// TwinCAT 3 PLC project PLC_Dev_Anker1
// ProgramVersion: 3.1.4024.0
// libraries:
//   EfficientIO Communicator, * (EfficientIO)
//   Tc2_Standard, * (Beckhoff Automation GmbH)
//   Tc2_System, * (Beckhoff Automation GmbH)
//   Tc3_Module, * (Beckhoff Automation GmbH)
// project tree:
//   DUTs/ struct_ADS_Anker.TcDUT
//   / FastTask.TcTTO, MiddleTask.TcTTO, SlowTask.TcTTO
//   FB/ FB_ADS_Read.TcPOU, F_AdsErrorText.TcPOU
//   POUs/ prgComEffIO.TcPOU, prgEM.TcPOU, prgEMS.TcPOU, prgRWEffIO.TcPOU, prgVarEffIO.TcPOU, prg_ADS.TcPOU
// (motion and I/O tree: see PLC project plc dev barac)
// real-time tasks:
//   TASK FastTask: cycle T#5ms, priority 19, ADS port 351
//   TASK SlowTask: cycle T#20ms, priority 22, ADS port 352
//   TASK MiddleTask: cycle T#10ms, priority 21, ADS port 353

CONFIGURATION PLC_Dev_Anker1
    RESOURCE PLC ON TwinCAT3
        TASK FastTask(INTERVAL := T#5ms, PRIORITY := 19);
        TASK MiddleTask(INTERVAL := T#10ms, PRIORITY := 21);
        TASK SlowTask(INTERVAL := T#20ms, PRIORITY := 22);
        PROGRAM prgRWEffIO WITH FastTask : prgRWEffIO;
        PROGRAM prgVarEffIO WITH FastTask : prgVarEffIO;
        PROGRAM prgEMS WITH MiddleTask : prgEMS;
        PROGRAM prgEM WITH MiddleTask : prgEM;
        PROGRAM prg_ADS WITH MiddleTask : prg_ADS;
        PROGRAM prgComEffIO WITH SlowTask : prgComEffIO;
    END_RESOURCE
END_CONFIGURATION

// ---- DUTs/struct_ADS_Anker.TcDUT
TYPE struct_ADS_Anker :
STRUCT
	int_liveCount		: INT;	
	
	// prgEM
	lr_RealPower_Grid			: LREAL;				
	lr_ApparentPower_Grid		: LREAL;				
	lr_ReactivePower_Grid		: LREAL;				
	lr_Frequency_Grid			: LREAL;				                                   
	lr_Voltage_L1N				: LREAL;				
	lr_Voltage_L2N				: LREAL;				
	lr_Voltage_L3N				: LREAL;				
	lr_Voltage_L1L2				: LREAL;				
	lr_Voltage_L2L3				: LREAL;				
	lr_Voltage_L3L1				: LREAL;				
 	lr_Current_L1				: LREAL;				
	lr_Current_L2				: LREAL;				
	lr_Current_L3				: LREAL;				
	lrPower_EM1					: LREAL;					
	lrPower_EM2					: LREAL;					
	lrPower_EM3					: LREAL;					
	lrPower_EM4					: LREAL;					
	lrPower_EM5					: LREAL;					
	lrPower_EM6					: LREAL;					
	lrPower_House				: LREAL;					
	lr_EnergyCounter_Grid		: LREAL;					
	lr_EnergyCounter_EM1		: LREAL;					
	lr_EnergyCounter_EM2		: LREAL;					
	lr_EnergyCounter_EM3		: LREAL;					
	lr_EnergyCounter_EM4		: LREAL;					
	lr_EnergyCounter_EM5		: LREAL;					
	lr_EnergyCounter_EM6		: LREAL;					
	lr_EnergyCounter_House		: LREAL;		

	// prgEMS
	b_Manual_On_CH1				: BOOL;						
	b_Manual_Off_CH1			: BOOL;						
	b_Manual_On_CH2				: BOOL;						
	b_Manual_Off_CH2			: BOOL;						
	b_Manual_On_CH3				: BOOL;						
	b_Manual_Off_CH3			: BOOL;						
	b_Manual_On_CH4				: BOOL;						
	b_Manual_Off_CH4			: BOOL;						
	b_Manual_On_CH5				: BOOL;						
	b_Manual_Off_CH5			: BOOL;						
	b_Manual_On_Coffee_CH6		: BOOL;				
	b_Manual_Off_Coffee_CH6		: BOOL;				
	b_Manual_On_Vent_CH7		: BOOL;				
	b_Manual_Off_Vent_CH7		: BOOL;			
	b_LoadOn_CH1				: BOOL;		
	b_LoadOn_CH2				: BOOL;			
	b_LoadOn_CH3				: BOOL;			
	b_LoadOn_CH4				: BOOL;			
	b_LoadOn_CH5				: BOOL;			
	b_LoadOn_CH6				: BOOL;			
	b_LoadOn_CH7				: BOOL;		
	byte_MoFr_Open_Hour			: BYTE;					
	byte_MoFr_Open_Minute		: BYTE;					
	byte_MoFr_Close_Hour		: BYTE;					
	byte_MoFr_Close_Minute		: BYTE;					
	byte_Sa_Open_Hour			: BYTE;					
	byte_Sa_Open_Minute			: BYTE;					
	byte_Sa_Close_Hour			: BYTE;					
	byte_Sa_Close_Minute		: BYTE;					
	byte_So_Open_Hour			: BYTE;					
	byte_So_Open_Minute			: BYTE;					
	byte_So_Close_Hour			: BYTE;					
	byte_So_Close_Minute		: BYTE;					
// offset CH1 in hours			                    
	b_Enable_Control_CH1		: BOOL;				
	real_Offset_Start_CH1		: REAL;				
	real_Offset_Stop_CH1		: REAL;				
// offset CH2 in hours			                    
	b_Enable_Control_CH2		: BOOL;				
	real_Offset_Start_CH2		: REAL;				
	real_Offset_Stop_CH2		: REAL;				
// offset CH3 in hours			                    
	b_Enable_Control_CH3		: BOOL;				
	real_Offset_Start_CH3		: REAL;				
	real_Offset_Stop_CH3		: REAL;				
// offset CH4 in hours			                    
	b_Enable_Control_CH4		: BOOL;				
	real_Offset_Start_CH4		: REAL;				
	real_Offset_Stop_CH4		: REAL;				
// offset CH5 in hours			                    
	b_Enable_Control_CH5		: BOOL;				
	real_Offset_Start_CH5		: REAL;				
	real_Offset_Stop_CH5		: REAL;				
// offset CH6 in hours			                    
	b_Enable_Control_Coffee_CH6	: BOOL;				
	real_Offset_Start_Coffee_CH6: REAL;				
	real_Offset_Stop_Coffee_CH6	: REAL;				
// offset CH7 in hours			                    
	b_Enable_Control_Vent_CH7	: BOOL;				
	real_Offset_Start_CH7		: REAL;				
	real_Offset_Stop_CH7		: REAL;				


                                  
			(*: REAL;			                        
			: REAL;                                     
			: REAL;			
			: REAL;			
			: REAL;
			: REAL;			
			: REAL;
			: REAL;			
*)

END_STRUCT
END_TYPE

// ---- POUs/prgRWEffIO.TcPOU
PROGRAM prgRWEffIO
VAR
	fbRW1		: FB_ReadWrite_V2;
END_VAR

fbRW1(eUploadType := eSelectDataUploadType.e_Change_Intervall5min, bBusy=> , bError=> , udiErrorCodeOut=> , eErrorReadWrite_Out=> );

END_PROGRAM

// ---- POUs/prgVarEffIO.TcPOU
PROGRAM prgVarEffIO
VAR
	fbVar		: FB_VarInfo_V3;
END_VAR

fbVar(
	bReadInfo:= , 
	eTMCFile:= eSelectTMCFile.eDontUseTMCFile, 
	eSavePositionTMCFile:= eSavePositionOnPLC.ePostionC, 
	udiCounterFoundVariables=> , 
	bError=> , 
	bBusy=> , 
	byProgress=> , 
	udiErrorCodeOut=> , 
	eErrorVarInfo_Out=> , 
	sVarWithError=> );

fbVar(
	bReadInfo:= , 
	eTMCFile:= eSelectTMCFile.eDontUseTMCFile, 
	eSavePositionTMCFile:= eSavePositionOnPLC.ePostionC,
	udiCounterFoundVariables=> , 
	bError=> , 
	bBusy=> , 
	byProgress=> , 
	udiErrorCodeOut=> , 
	eErrorVarInfo_Out=> , 
	sVarWithError=> );
	
fbVar(
	bReadInfo:= , 
	eTMCFile:= eSelectTMCFile.eDontUseTMCFile, 
	eSavePositionTMCFile:= eSavePositionOnPLC.ePostionC,
	udiCounterFoundVariables=> , 
	bError=> , 
	bBusy=> , 
	byProgress=> , 
	udiErrorCodeOut=> , 
	eErrorVarInfo_Out=> , 
	sVarWithError=> );

END_PROGRAM

// ---- POUs/prgEMS.TcPOU
PROGRAM prgEMS
VAR	
	b_Manual_On_CH1		: BOOL;						//{#lynus.ag#()}
	b_Manual_Off_CH1	: BOOL;						//{#lynus.ag#()}
	b_Manual_On_CH2		: BOOL;						//{#lynus.ag#()}
	b_Manual_Off_CH2	: BOOL;						//{#lynus.ag#()}
	b_Manual_On_CH3		: BOOL;						//{#lynus.ag#()}
	b_Manual_Off_CH3	: BOOL;						//{#lynus.ag#()}
	b_Manual_On_CH4		: BOOL;						//{#lynus.ag#()}
	b_Manual_Off_CH4	: BOOL;						//{#lynus.ag#()}
	b_Manual_On_CH5		: BOOL;						//{#lynus.ag#()}
	b_Manual_Off_CH5	: BOOL;						//{#lynus.ag#()}
	b_Manual_On_Coffee_CH6		: BOOL;						//{#lynus.ag#()}
	b_Manual_Off_Coffee_CH6		: BOOL;						//{#lynus.ag#()}
	b_Manual_On_Vent_CH7		: BOOL;						//{#lynus.ag#()}
	b_Manual_Off_Vent_CH7		: BOOL;						//{#lynus.ag#()}
	mtest: BOOL;

	b_LoadOn_CH1	: BOOL;						//{#lynus.ag#()}
	b_LoadOn_CH2	: BOOL;						//{#lynus.ag#()}
	b_LoadOn_CH3	: BOOL;						//{#lynus.ag#()}
	b_LoadOn_CH4	: BOOL;						//{#lynus.ag#()}
	b_LoadOn_CH5	: BOOL;						//{#lynus.ag#()}
	b_LoadOn_CH6	: BOOL;						//{#lynus.ag#()}
	b_LoadOn_CH7	: BOOL;						//{#lynus.ag#()}
	b_Input_KeySwitch		: BOOL;						//{#lynus.ag#()}
	b_Input_Spare			: BOOL;						//{#lynus.ag#()}
	m_UnderGroundMode		: BOOL;						//{#lynus.ag#()}
// opening hours
	byte_MoFr_Open_Hour		:BYTE;					//{#lynus.ag#()}
	byte_MoFr_Open_Minute	:BYTE;					//{#lynus.ag#()}
	byte_MoFr_Close_Hour	:BYTE;					//{#lynus.ag#()}
	byte_MoFr_Close_Minute	:BYTE;					//{#lynus.ag#()}
	byte_Sa_Open_Hour		:BYTE;					//{#lynus.ag#()}
	byte_Sa_Open_Minute		:BYTE;					//{#lynus.ag#()}
	byte_Sa_Close_Hour		:BYTE;					//{#lynus.ag#()}
	byte_Sa_Close_Minute	:BYTE;					//{#lynus.ag#()}
	byte_So_Open_Hour		:BYTE;					//{#lynus.ag#()}
	byte_So_Open_Minute		:BYTE;					//{#lynus.ag#()}
	byte_So_Close_Hour		:BYTE;					//{#lynus.ag#()}
	byte_So_Close_Minute	:BYTE;					//{#lynus.ag#()}
// offset CH1 in hours			
	b_Enable_Control_CH1		:BOOL;				//{#lynus.ag#()}
	real_Offset_Start_CH1		:REAL;				//{#lynus.ag#()}
	real_Offset_Stop_CH1		:REAL;				//{#lynus.ag#()}
// offset CH2 in hours			
	b_Enable_Control_CH2		:BOOL;				//{#lynus.ag#()}
	real_Offset_Start_CH2		:REAL;				//{#lynus.ag#()}
	real_Offset_Stop_CH2		:REAL;				//{#lynus.ag#()}
// offset CH3 in hours			
	b_Enable_Control_CH3		:BOOL;				//{#lynus.ag#()}
	real_Offset_Start_CH3		:REAL;				//{#lynus.ag#()}
	real_Offset_Stop_CH3		:REAL;				//{#lynus.ag#()}
// offset CH4 in hours			
	b_Enable_Control_CH4		:BOOL;				//{#lynus.ag#()}
	real_Offset_Start_CH4		:REAL;				//{#lynus.ag#()}
	real_Offset_Stop_CH4		:REAL;				//{#lynus.ag#()}
// offset CH5 in hours			
	b_Enable_Control_CH5		:BOOL;				//{#lynus.ag#()}
	real_Offset_Start_CH5		:REAL;				//{#lynus.ag#()}
	real_Offset_Stop_CH5		:REAL;				//{#lynus.ag#()}
// offset CH6 in hours			
	b_Enable_Control_Coffee_CH6	:BOOL;				//{#lynus.ag#()}
	real_Offset_Start_Coffee_CH6:REAL;				//{#lynus.ag#()}
	real_Offset_Stop_Coffee_CH6	:REAL;				//{#lynus.ag#()}
// offset CH7 in hours			
	b_Enable_Control_Vent_CH7	:BOOL;				//{#lynus.ag#()}
	real_Offset_Start_CH7		:REAL;				//{#lynus.ag#()}
	real_Offset_Stop_CH7		:REAL;				//{#lynus.ag#()}
END_VAR

b_Manual_On_CH1	:=	prg_ADS.struct_received.b_Manual_On_CH1	;
b_Manual_Off_CH1	:=	prg_ADS.struct_received.b_Manual_Off_CH1	;
b_Manual_On_CH2	:=	prg_ADS.struct_received.b_Manual_On_CH2	;
b_Manual_Off_CH2	:=	prg_ADS.struct_received.b_Manual_Off_CH2	;
b_Manual_On_CH3	:=	prg_ADS.struct_received.b_Manual_On_CH3	;
b_Manual_Off_CH3	:=	prg_ADS.struct_received.b_Manual_Off_CH3	;
b_Manual_On_CH4	:=	prg_ADS.struct_received.b_Manual_On_CH4	;
b_Manual_Off_CH4	:=	prg_ADS.struct_received.b_Manual_Off_CH4	;
b_Manual_On_CH5	:=	prg_ADS.struct_received.b_Manual_On_CH5	;
b_Manual_Off_CH5	:=	prg_ADS.struct_received.b_Manual_Off_CH5	;
b_Manual_On_Coffee_CH6	:=	prg_ADS.struct_received.b_Manual_On_Coffee_CH6	;
b_Manual_Off_Coffee_CH6	:=	prg_ADS.struct_received.b_Manual_Off_Coffee_CH6	;
b_Manual_On_Vent_CH7	:=	prg_ADS.struct_received.b_Manual_On_Vent_CH7	;
b_Manual_Off_Vent_CH7	:=	prg_ADS.struct_received.b_Manual_Off_Vent_CH7	;
b_LoadOn_CH1	:=	prg_ADS.struct_received.b_LoadOn_CH1	;
b_LoadOn_CH2	:=	prg_ADS.struct_received.b_LoadOn_CH2	;
b_LoadOn_CH3	:=	prg_ADS.struct_received.b_LoadOn_CH3	;
b_LoadOn_CH4	:=	prg_ADS.struct_received.b_LoadOn_CH4	;
b_LoadOn_CH5	:=	prg_ADS.struct_received.b_LoadOn_CH5	;
b_LoadOn_CH6	:=	prg_ADS.struct_received.b_LoadOn_CH6	;
b_LoadOn_CH7	:=	prg_ADS.struct_received.b_LoadOn_CH7	;
byte_MoFr_Open_Hour	:=	prg_ADS.struct_received.byte_MoFr_Open_Hour	;
byte_MoFr_Open_Minute	:=	prg_ADS.struct_received.byte_MoFr_Open_Minute	;
byte_MoFr_Close_Hour	:=	prg_ADS.struct_received.byte_MoFr_Close_Hour	;
byte_MoFr_Close_Minute	:=	prg_ADS.struct_received.byte_MoFr_Close_Minute	;
byte_Sa_Open_Hour	:=	prg_ADS.struct_received.byte_Sa_Open_Hour	;
byte_Sa_Open_Minute	:=	prg_ADS.struct_received.byte_Sa_Open_Minute	;
byte_Sa_Close_Hour	:=	prg_ADS.struct_received.byte_Sa_Close_Hour	;
byte_Sa_Close_Minute	:=	prg_ADS.struct_received.byte_Sa_Close_Minute	;
byte_So_Open_Hour	:=	prg_ADS.struct_received.byte_So_Open_Hour	;
byte_So_Open_Minute	:=	prg_ADS.struct_received.byte_So_Open_Minute	;
byte_So_Close_Hour	:=	prg_ADS.struct_received.byte_So_Close_Hour	;
byte_So_Close_Minute	:=	prg_ADS.struct_received.byte_So_Close_Minute	;
b_Enable_Control_CH1	:=	prg_ADS.struct_received.b_Enable_Control_CH1	;
real_Offset_Start_CH1	:=	prg_ADS.struct_received.real_Offset_Start_CH1	;
real_Offset_Stop_CH1	:=	prg_ADS.struct_received.real_Offset_Stop_CH1	;
b_Enable_Control_CH2	:=	prg_ADS.struct_received.b_Enable_Control_CH2	;
real_Offset_Start_CH2	:=	prg_ADS.struct_received.real_Offset_Start_CH2	;
real_Offset_Stop_CH2	:=	prg_ADS.struct_received.real_Offset_Stop_CH2	;
b_Enable_Control_CH3	:=	prg_ADS.struct_received.b_Enable_Control_CH3	;
real_Offset_Start_CH3	:=	prg_ADS.struct_received.real_Offset_Start_CH3	;
real_Offset_Stop_CH3	:=	prg_ADS.struct_received.real_Offset_Stop_CH3	;
b_Enable_Control_CH4	:=	prg_ADS.struct_received.b_Enable_Control_CH4	;
real_Offset_Start_CH4	:=	prg_ADS.struct_received.real_Offset_Start_CH4	;
real_Offset_Stop_CH4	:=	prg_ADS.struct_received.real_Offset_Stop_CH4	;
b_Enable_Control_CH5	:=	prg_ADS.struct_received.b_Enable_Control_CH5	;
real_Offset_Start_CH5	:=	prg_ADS.struct_received.real_Offset_Start_CH5	;
real_Offset_Stop_CH5	:=	prg_ADS.struct_received.real_Offset_Stop_CH5	;
b_Enable_Control_Coffee_CH6	:=	prg_ADS.struct_received.b_Enable_Control_Coffee_CH6	;
real_Offset_Start_Coffee_CH6	:=	prg_ADS.struct_received.real_Offset_Start_Coffee_CH6	;
real_Offset_Stop_Coffee_CH6	:=	prg_ADS.struct_received.real_Offset_Stop_Coffee_CH6	;
b_Enable_Control_Vent_CH7	:=	prg_ADS.struct_received.b_Enable_Control_Vent_CH7	;
real_Offset_Start_CH7	:=	prg_ADS.struct_received.real_Offset_Start_CH7	;
real_Offset_Stop_CH7	:=	prg_ADS.struct_received.real_Offset_Stop_CH7	;

END_PROGRAM

// ---- POUs/prg_ADS.TcPOU
PROGRAM prg_ADS
VAR
	ADS_1: FB_ADS_Read;
	str_ADS_read: STRING(40);
	byte_array : ARRAY[0..1023] OF BYTE;
	struct_received	: struct_ADS_Anker;						
	int_liveCount		: INT;						//{#lynus.ag#()}
	byte_old: BYTE;
END_VAR


str_ADS_read := 'prgComEffIO.byte_array';

ADS_1(
	udintWriteLength:=  SIZEOF(byte_array), 
	udintReadLength:= SIZEOF(byte_array), 
	dwSourceAddr:= ADR(str_ADS_read), 
	dwDestAddr:= ADR(byte_array), 
	strNetID:= '5.146.122.188.1.1', // EIOAN010009 Meidlinger Hauptstraße 77-79 Meidlinger Hauptstraße 77-79        Filiale 5261
	timeReadDelay:= T#5S, 
	mADSError=> , 
	strADSErrorText=> );
	
// copy struct to byte array
IF byte_array[1] <> byte_old AND NOT ADS_1.mADSError AND byte_array[1] <> 0 THEN
	IF SIZEOF(struct_received) > SIZEOF(byte_array) THEN
		memcpy(ADR(struct_received),ADR(byte_array),SIZEOF(byte_array));
	ELSE
		memcpy(ADR(struct_received),ADR(byte_array),SIZEOF(struct_received));
	END_IF
	byte_old := byte_array[1];
END_IF
	
	
int_liveCount := prg_ADS.struct_received.int_liveCount 	;

END_PROGRAM

// ---- FB/FB_ADS_Read.TcPOU
FUNCTION_BLOCK FB_ADS_Read
VAR
	intState: INT;
	fbADSRDWRT: ADSRDWRT;
	Timer1: TON;
END_VAR
VAR_INPUT
	udintWriteLength:UDINT;
	udintReadLength:UDINT;
	dwSourceAddr:pvoid;
	dwDestAddr:PVOID;
	strNetID: STRING;
	timeReadDelay:TIME;
END_VAR
VAR_OUTPUT
	mADSError: BOOL;
	strADSErrorText: STRING;
END_VAR

timeReadDelay := LIMIT(T#100MS,timeReadDelay,T#24H);

CASE intState OF
	0:	(* start reading *)
		fbADSRDWRT.WRITELEN:=udintWriteLength;
		fbADSRDWRT.READLEN:=udintReadLength;
		fbADSRDWRT.SRCADDR:=dwSourceAddr;
		fbADSRDWRT.DESTADDR:=dwDestAddr;
		fbADSRDWRT.WRTRD:=TRUE;
		intState:=1000;
	1000: (* wait for reply *)
		IF NOT fbADSRDWRT.BUSY THEN
			fbADSRDWRT.WRTRD:=FALSE;
			IF NOT fbADSRDWRT.ERR THEN
				strADSErrorText:='no error';
				mADSError:=FALSE;
				Timer1.IN:=TRUE;
				intState:=1100;
			ELSE
				strADSErrorText:=F_AdsErrorText(fbADSRDWRT.ERRID);
				mADSError:=TRUE;
				Timer1.IN:=TRUE;
				intState:=1100;
			END_IF
		END_IF
	1100: (* wait to hold state *)
		fbADSRDWRT.WRTRD:=FALSE;
		IF Timer1.Q THEN
			Timer1.IN:=FALSE;
			intState:=0;
		END_IF
		
END_CASE

Timer1(PT:=timeReadDelay);


fbADSRDWRT(
	NETID:=strNetID,
	PORT:=851,
	IDXGRP:=16#F004,
	IDXOFFS:=0,
	TMOUT:=t#10s);


(*
VAR_INPUT
        NETID           : T_AmsNetId;
        PORT            : T_AmsPort;
        IDXGRP          : UDINT;
        IDXOFFS         : UDINT;
        WRITELEN                : UDINT;
        READLEN         : UDINT;
        SRCADDR                 : DWORD;
        DESTADDR                : DWORD;
        WRTRD           : BOOL;
        TMOUT           : TIME;
END_VAR
VAR_OUTPUT
        BUSY            : BOOL;
        ERR             : BOOL;
        ERRID           : UDINT;
END_VAR

*)

END_FUNCTION_BLOCK

// ---- FB/F_AdsErrorText.TcPOU
FUNCTION F_AdsErrorText : STRING
VAR_INPUT
	nAdsError:UDINT;
END_VAR
VAR
	sText:STRING(255);
END_VAR

(*
ADS Return Codes

Fehlernummern: 0x000..., 0x500..., 0x700..., 0x1000..., 0x274C...

Global Error Codes

Hex Dez Beschreibung 
0x0 0 kein Fehler 
0x1 1 Internal error 
0x2 2 No Rtime 
0x3 3 Allocation locked memory error 
0x4 4 Insert mailbox error 
0x5 5 Wrong receive HMSG 
0x6 6 target port not found 
0x7 7 target machine not found 
0x8 8 Unknown command ID 
0x9 9 Bad task ID 
0xA 10 No IO 
0xB 11 Unknown AMS command 
0xC 12 Win 32 error 
0xD 13 Port not connected 
0xE 14 Invalid AMS length 
0xF 15 Invalid AMS Net ID 
0x10 16 Low Installation level 
0x11 17 No debug available 
0x12 18 Port disabled 
0x13 19 Port already connected 
0x14 20 AMS Sync Win32 error 
0x15 21 AMS Sync Timeout 
0x16 22 AMS Sync AMS error 
0x17 23 AMS Sync no index map 
0x18 24 Invalid AMS port 
0x19 25 No memory 
0x1A 26 TCP send error 
0x1B 27 Host unreachable 

 

Router Error Codes

Hex Dez Fehlertyp Beschreibung 
0x500 1280 Intern ROUTERERR_NOLOCKEDMEMORY
Es konnte kein nicht auslagerbarer Speicher alloziert werden. 
0x501  1281  Intern  ROUTERERR_RESIZEMEMORY
Der Routerspeicher konnte nicht in seiner Größe verändert werden.  
0x502  1282  Intern  ROUTERERR_MAILBOXFULL
Die Mailbox eines AmsPorts hat die maximal mögliche Anzahl Einträge erreicht.
Die aktuell gesendete Nachricht wurde verworfen.  
0x503  1283  Intern  ROUTERERR_DEBUGBOXFULL
Die Mailbox des Ams Debugger Ports  hat die maximal mögliche Anzahl Einträge erreicht.
Die gesendete Nachricht wird nicht im Debug Monitor angezeigt.  
0x504  1284  Intern  ROUTERERR_UNKNOWNPORTTYPE   
0x505  1285  Intern  ROUTERERR_NOTINITIALIZED
Router ist (noch) nicht initialisiert.  
0x506  1286  Intern  ROUTERERR_PORTALREADYINUSE 
Die gewünschte Portnummer ist schon vergeben.  
0x507  1287  Intern  ROUTERERR_NOTREGISTERED 
Ams Port ist nicht registriert.  
0x508  1288  Intern  ROUTERERR_NOMOREQUEUES
Die maximale Anzahl möglicher Ams Ports ist erreicht.  
0x509  1289  Intern  ROUTERERR_INVALIDPORT   
0x50A  1290  Intern  ROUTERERR_NOTACTIVATED 
Der TwinCAT Router ist (noch) nicht aktiv.  

 

General ADS Error Codes

Hex Dez Beschreibung 
0x700 1792 error class <device error> 
0x701 1793 Service is not supported by server 
0x702 1794 invalid index group 
0x703 1795 invalid index offset 
0x704 1796 reading/writing not permitted 
0x705 1797  parameter size not correct 
0x706 1798 invalid parameter value(s) 
0x707 1799 device is not in a ready state 
0x708 1800 device is busy 
0x709 1801 invalid context (must be in Windows) 
0x70A 1802 out of memory 
0x70B 1803 invalid parameter value(s) 
0x70C 1804 not found (files, ...) 
0x70D 1805 syntax error in command or file 
0x70E 1806 objects do not match 
0x70F 1807 object already exists 
0x710 1808 symbol not found 
0x711 1809 symbol version invalid 
0x712 1810 server is in invalid state 
0x713 1811 AdsTransMode not supported 
0x714 1812 Notification handle is invalid 
0x715 1813 Notification client not registered 
0x716 1814 no more notification handles 
0x717 1815 size for watch too big 
0x718 1816 device not initialized 
0x719 1817 device has a timeout 
0x71A 1818 query interface failed 
0x71B 1819 wrong interface required 
0x71C 1820 class ID is invalid 
0x71D 1821 object ID is invalid 
0x71E 1822 request is pending 
0x71F 1823 request is aborted 
0x720 1824 signal warning 
0x721 1825 invalid array index 
0x722 1826 symbol not active -> release handle and try again 
0x723 1827 access denied 
0x740 1856 Error class <client error> 
0x741 1857 invalid parameter at service 
0x742 1858 polling list is empty 
0x743 1859 var connection already in use 
0x744 1860 invoke ID in use 
0x745 1861 timeout elapsed 
0x746 1862 error in win32 subsystem 
0x748 1864 ads port not opened 
0x750 1872 internal error in ads sync 
0x751 1873 hash table overflow 
0x752 1874 key not found in hash 
0x753 1875 no more symbols in cache 
0x754 1876 invalid response received 
0x755 1877 Sync port locked
ADS-Client tries to send a ADS msg but another thread is still waiting for an ADS-response. 
This error occurs only if no ADS-router is installed (please install royalty free TwinCAT-CP) 
or the router does not know the remote ADS device (define the remote ADS partner ) 

 

RTime Error Codes

Hex Dez Fehlertyp Beschreibung 
0x1000  4096  Intern  RTERR_INTERNAL 
Interner fataler Fehler im TwinCAT Echtzeitsystem  
0x1001  4097  Intern  RTERR_BADTIMERPERIODS
Ungültiger Timerwert.  
0x1002  4098  Intern  RTERR_INVALIDTASKPTR
Task Pointer hat den ungültigen Wert NULL.  
0x1003  4099  Intern  RTERR_INVALIDSTACKPTR
Task Stack Pointer hat den ungültigen Wert NULL.  
0x1004  4100  Intern  RTERR_PRIOEXISTS
Die geforderte Taskpriorität ist schon vergeben.  
0x1005  4101  Intern  RTERR_NOMORETCB
Kein freier TCB (Task Control Block) mehr verfügbar. Maximale Anzahl von TCBs ist 64.  
0x1006  4102  Intern  RTERR_NOMORESEMAS
Keine freie Semaphore mehr verfügbar. Maximale Anzahl von Semaphoren ist 64.  
0x1007  4103  Intern  RTERR_NOMOREQUEUES
Keine freie Queue mehr verfügbar. Maximale Anzahl von Queues ist 64.  
0x1008  4104  Intern  TwinCAT reserved.  
0x1009  4105  Intern  TwinCAT reserved.  
0x100A  4106  Intern  TwinCAT reserved.  
0x100B  4107  Intern  TwinCAT reserved.  
0x100C 4108  Intern  TwinCAT reserved.  
0x100D 4109  Intern  RTERR_EXTIRQALREADYDEF
Ein externer Synchronisierungsinterrupt ist schon angemeldet.  
0x100E 4110  Intern  RTERR_EXTIRQNOTDEF
Kein externer Synchronisierungsinterrupt angemeldet.  
0x100F 4111  Intern  RTERR_EXTIRQINSTALLFAILED
Anmelden des externen Synchronisierungsinterrupts ist fehlgeschlagen.  
0x1010  4112  Intern  RTERR_IRQLNOTLESSOREQUAL
Aufruf einer Dienstfunktion im falschen Kontext.  

 

Socket Error Codes

Hex Dez Beschreibung 
0x274c 10060 A socket operation was attempted to an unreachable host 
0x274d 10061 A connection attempt failed because the connected party did not properly respond after a period of time, 
or established connection failed because connected host has failed to respond. 
0x2751 10065 No connection could be made because the target machine actively refused it 
    Weitere Socket Fehler-Codes finden Sie hier: Win32 Error Codes 

*)

CASE nAdsError OF
	0	:		sText := 'kein Fehler';
	1	:		sText := 'Internal error';
	2	:		sText := 'No Rtime';
	3	:		sText := 'Allocation locked memory error';
	4	:		sText := 'Insert mailbox error';
	5	:		sText := 'Wrong receive HMSG';
	6	:		sText := 'target port not found';
	7	:		sText := 'target machine not found';
	8	:		sText := 'Unknown command ID';
	9	:		sText := 'Bad task ID';
	10	:		sText := 'No IO';
	11	:		sText := 'Unknown AMS command';
	12	:		sText := 'Win 32 error';
	13	:		sText := 'Port not connected';
	14	:		sText := 'Invalid AMS length';
	15	:		sText := 'Invalid AMS Net ID';
	16	:		sText := 'Low Installation level';
	17	:		sText := 'No debug available';
	18	:		sText := 'Port disabled';
	19	:		sText := 'Port already connected';
	20	:		sText := 'AMS Sync Win32 error';
	21	:		sText := 'AMS Sync Timeout';
	22	:		sText := 'AMS Sync AMS error';
	23	:		sText := 'AMS Sync no index map';
	24	:		sText := 'Invalid AMS port';
	25	:		sText := 'No memory ';
	26	:		sText := 'TCP send error ';
	27	:		sText := 'Host unreachable';
	1280	:		sText := 'Router: no locked memory ';
	1282	:		sText := 'Router: mailbox full ';
	1792	:		sText := 'error class <device error> ';
	1793	:		sText := 'Service is not supported by server ';
	1794	:		sText := 'invalid index group ';
	1795	:		sText := 'invalid index offset ';
	1796	:		sText := 'reading-writing not permitted ';
	1797	:		sText:='parameter size not correct';
	1798	:		sText := 'invalid parameter value ';
	1799	:		sText := 'device is not in a ready state ';
	1800	:		sText := 'device is busy ';
	1801	:		sText := 'invalid context (must be in Windows) ';
	1802	:		sText := 'out of memory';
	1803	:		sText := 'invalid parameter value(s)';
	1804	:		sText := 'not found (files, ...)';
	1805	:		sText := 'syntax error in command or file';
	1806	:		sText := 'objects do not match';
	1807	:		sText := 'object already exists';
	1808	:		sText := 'symbol not found';
	1809	:		sText := 'symbol version invalid';
	1810	:		sText := 'server is in invalid state';
	1811	:		sText := 'AdsTransMode not supported';
	1812	:		sText := 'Notification handle is invalid';
	1813	:		sText := 'Notification client not registered';
	1814	:		sText := 'no more notification handles';
	1815	:		sText := 'size for watch too big';
	1816	:		sText := 'device not initialized';
	1817	:		sText := 'device has a timeout';
	1818	:		sText := 'query interface failed';
	1819	:		sText := 'wrong interface required';
	1820	:		sText := 'class ID is invalid';
	1821	:		sText := 'object ID is invalid';
	1822	:		sText := 'request is pending';
	1823	:		sText := 'request is aborted';
	1824	:		sText := 'signal warning';
	1825	:		sText := 'invalid array index';
	1856	:		sText := 'Error class <client error>';
	1857	:		sText := 'invalid parameter at service';
	1858	:		sText := 'polling list is empty';
	1859	:		sText := 'var connection already in use';
	1860	:		sText := 'invoke ID in use';
	1861	:		sText := 'timeout elapsed';
	1862	:		sText := 'error in win32 subsystem';
	1864	:		sText := 'ads port not opened';
	1872	:		sText := 'internal error in ads sync';
	1873	:		sText := 'hash table overflow';
	1874	:		sText := 'key not found in hash';
	1875	:		sText := 'no more symbols in cache';
	1877	:		sText := 'Sync port locked: ADS-Client tries to send a ADS msg but another thread is still waiting for an ADS-response. This error occurs only if no ADS-router is installed or the router does not know the remote ADS device (define the remote ADS partner )';
	10060	:		sText := 'A socket operation was attempted to an unreachable host';
	10061	:		sText := 'A connection attempt failed because the connected party did not properly respond after a period of time, or established connection failed because connected host has failed to respond.';
	10065	:		sText := 'No connection could be made because the target machine actively refused it';

(* FB_SmtpV2 *)
	32778 	:	sText := 'Not connected';
	32779 	:	sText := 'Sender expected';
	32780 	:	sText := 'Recipients expected';
	32781 	:	sText := 'Send FROM command failed';
	32782 	:	sText := 'Send DATA command failed';
	32783 	:	sText := 'Send mail header failed';
	32784 	:	sText := 'Send mail body failed';
	32785 	:	sText := 'Send "end of mail indicator" failed';
	32786 	:	sText := 'Send "RCPT" command failed';
	32787 	:	sText := 'Server Response got no username request';
	32788 	:	sText := 'Server Response got no password request';
	32789 	:	sText := 'Unable to create socket connection';
	32790 	:	sText := 'Authentication type not supported by smtp server';
	32791 	:	sText := 'Wrong username or password';
	32792 	:	sText := 'Not supported';
	32793 	:	sText := 'Invalid hostname';
	32794 	:	sText := 'Unable to send attachment';
	32795 	:	sText := 'File not found';
	32796 	:	sText := 'Invalid Version (New SMTP Server with old SMTP PLC library)';
	32797 	:	sText := 'Unable to connect (Connection error => sometimes wrong port or wrong server)';
	32798 	:	sText := 'Unable to create socket';
	32799 	:	sText := 'WSA startup failed';
	32800 	:	sText := 'Invalid hostname';
	32801 	:	sText := 'Unecpected response from server';
	32802 	:	sText := 'Error while receiving data';
	32803 	:	sText := 'No supported authentication methods found';
	32804 	:	sText := 'Invalid parameter';
	32928 	:	sText := 'Security interface not found';
	32929 	:	sText := 'Unable to call security interface';
	32930 	:	sText := 'Security initialization failed';
	32932 	:	sText := 'Unable to create credentials';
	32933 	:	sText := 'SSL-handshake failed';
	32934 	:	sText := 'Invalid server credentials';
	32935 	:	sText := 'Unable to verify server';
	32936 	:	sText := 'Unable to encrypt message';
	32937 	:	sText := 'Unable to decrypt message';


	ELSE			sText := 'Error not defined';
END_CASE;

F_ADSerrorText := sText;

END_FUNCTION

// ---- POUs/prgComEffIO.TcPOU
PROGRAM prgComEffIO
VAR
	fbCom		: FB_MqttCommunicator_v3;

END_VAR

fbCom(
	bConnect:= TRUE, 
	strAuthkey := 'DEV01673741737',
	sUserName:= '42cf3b23-700d-4275-a072-1301ce2666ee' , 		
	sUserPassword:= 'abe4fa5d-8e50-48f0-873c-207b5a84d6b6',
	eSavePositionCertificate:= eSavePositionOnPLC.ePostionC, 
	bConnected=> , 
	bError=> , 
	hrErrorCode=> , 
	eConnectionState=> , 
	eErrorMessage_Out=> );

END_PROGRAM

// ---- POUs/prgEM.TcPOU
PROGRAM prgEM
VAR
	lr_RealPower_Grid	: LREAL;						//{#lynus.ag#()}
	lr_ApparentPower_Grid: LREAL;						//{#lynus.ag#()}
	lr_ReactivePower_Grid: LREAL;						//{#lynus.ag#()}
	lr_Frequency_Grid	: LREAL;						//{#lynus.ag#()}
	lr_Voltage_L1N		: LREAL;						//{#lynus.ag#()}
	lr_Voltage_L2N		: LREAL;						//{#lynus.ag#()}
	lr_Voltage_L3N		: LREAL;						//{#lynus.ag#()}
	lr_Voltage_L1L2		: LREAL;						//{#lynus.ag#()}
	lr_Voltage_L2L3		: LREAL;						//{#lynus.ag#()}
	lr_Voltage_L3L1		: LREAL;						//{#lynus.ag#()}
 	lr_Current_L1		: LREAL;						//{#lynus.ag#()}
	lr_Current_L2		: LREAL;						//{#lynus.ag#()}
	lr_Current_L3		: LREAL;						//{#lynus.ag#()}
	lrPower_EM1		: LREAL;						//{#lynus.ag#()}
	lrPower_EM2		: LREAL;						//{#lynus.ag#()}
	lrPower_EM3		: LREAL;						//{#lynus.ag#()}
	lrPower_EM4		: LREAL;						//{#lynus.ag#()}
	lrPower_EM5		: LREAL;						//{#lynus.ag#()}
	lrPower_EM6		: LREAL;						//{#lynus.ag#()}
	lrPower_House	: LREAL;						//{#lynus.ag#()}
	lr_EnergyCounter_Grid	: LREAL;						//{#lynus.ag#()}
	lr_EnergyCounter_EM1	: LREAL;						//{#lynus.ag#()}
	lr_EnergyCounter_EM2	: LREAL;						//{#lynus.ag#()}
	lr_EnergyCounter_EM3	: LREAL;						//{#lynus.ag#()}
	lr_EnergyCounter_EM4	: LREAL;						//{#lynus.ag#()}
	lr_EnergyCounter_EM5	: LREAL;						//{#lynus.ag#()}
	lr_EnergyCounter_EM6	: LREAL;						//{#lynus.ag#()}
	lr_EnergyCounter_House	: LREAL;						//{#lynus.ag#()}
END_VAR

lr_RealPower_Grid		:=		prg_ADS.struct_received.lr_RealPower_Grid	;
lr_ApparentPower_Grid		:=		prg_ADS.struct_received.lr_ApparentPower_Grid	;
lr_ReactivePower_Grid		:=		prg_ADS.struct_received.lr_ReactivePower_Grid	;
lr_Frequency_Grid		:=		prg_ADS.struct_received.lr_Frequency_Grid	;
lr_Voltage_L1N		:=		prg_ADS.struct_received.lr_Voltage_L1N	;
lr_Voltage_L2N		:=		prg_ADS.struct_received.lr_Voltage_L2N	;
lr_Voltage_L3N		:=		prg_ADS.struct_received.lr_Voltage_L3N	;
lr_Voltage_L1L2		:=		prg_ADS.struct_received.lr_Voltage_L1L2	;
lr_Voltage_L2L3		:=		prg_ADS.struct_received.lr_Voltage_L2L3	;
lr_Voltage_L3L1		:=		prg_ADS.struct_received.lr_Voltage_L3L1	;
lr_Current_L1		:=		prg_ADS.struct_received.lr_Current_L1	;
lr_Current_L2		:=		prg_ADS.struct_received.lr_Current_L2	;
lr_Current_L3		:=		prg_ADS.struct_received.lr_Current_L3	;
lrPower_EM1		:=		prg_ADS.struct_received.lrPower_EM1	;
lrPower_EM2		:=		prg_ADS.struct_received.lrPower_EM2	;
lrPower_EM3		:=		prg_ADS.struct_received.lrPower_EM3	;
lrPower_EM4		:=		prg_ADS.struct_received.lrPower_EM4	;
lrPower_EM5		:=		prg_ADS.struct_received.lrPower_EM5	;
lrPower_EM6		:=		prg_ADS.struct_received.lrPower_EM6	;
lrPower_House		:=		prg_ADS.struct_received.lrPower_House	;
lr_EnergyCounter_Grid		:=		prg_ADS.struct_received.lr_EnergyCounter_Grid	;
lr_EnergyCounter_EM1		:=		prg_ADS.struct_received.lr_EnergyCounter_EM1	;
lr_EnergyCounter_EM2		:=		prg_ADS.struct_received.lr_EnergyCounter_EM2	;
lr_EnergyCounter_EM3		:=		prg_ADS.struct_received.lr_EnergyCounter_EM3	;
lr_EnergyCounter_EM4		:=		prg_ADS.struct_received.lr_EnergyCounter_EM4	;
lr_EnergyCounter_EM5		:=		prg_ADS.struct_received.lr_EnergyCounter_EM5	;
lr_EnergyCounter_EM6		:=		prg_ADS.struct_received.lr_EnergyCounter_EM6	;
lr_EnergyCounter_House		:=		prg_ADS.struct_received.lr_EnergyCounter_House	;

END_PROGRAM
